(* CODESYS project contpiezasfun.project
   CustomField01_name: CustomField01
   CustomField08_name: CustomField08
   CustomField06_name: CustomField06
   Title: ATV_IMC_Template
   CustomField09_name: CustomField09
   CustomField07_name: CustomField07
   CustomField05_name: CustomField05
   Author: sergi gomez
   CustomField02_name: CustomField02
   Description: This template can be used for a correct interface with the local drive. the MANDATORY_AT_EACH_CYCLE program must be called like it is done in this application.
   CustomField04_name: CustomField04
   CustomField10_name: CustomField10
   Version: 0.0.0.0
   Company: Schneider Electric
   CustomField03_name: CustomField03

Project tree, tasks and I/O mapping:
  MyController : TM241CE24R, Schneider Electric, order no. TM241CE24R, version 4.0.2.9
    application Application
      task MAST (cyclic, interval 20 ms, priority 15, watchdog 100 ms x 1) calls progpiezas
      function HiddenPOU [ST]
      global variables GVL
      program progpiezas [LD]
      visualisation scada
    DI : Digital Inputs, Schneider Electric, version 4.0.2.9
        input  iwDI_IW0 : WORD  // IW0
        input  Application.progpiezas.sensorcil : BOOL  // IW0.I0
        input  Application.progpiezas.almacenaje : BOOL  // IW0.I1
        input  ibDI_IB1 : BYTE  // IB1
    DQ : Digital Outputs, Schneider Electric, version 4.0.2.9
        output qwDQ_QW0 : WORD  // QW0
        output qbDQ_QB1 : BYTE  // QB1
    Counters : Counters, Schneider Electric, version 4.0.2.9
    Pulse_Generators : Pulse Generators, Schneider Electric, version 4.0.2.9
    Cartridge_1 : Cartridge, Schneider Electric, version 4.0.2.9
    IO_Bus : IO bus - TM3, Schneider Electric, version 4.0.2.9
      Module_1 : TM3DQ8R/G, Schneider Electric, order no. TM3DQ8R/G, version 1.0.1.3
          output Application.progpiezas.contpiezas.cilrec : BOOL  // QB0.Q0
          output Application.progpiezas.contpiezas.cilext : BOOL  // QB0.Q1
          output Application.cinta : BOOL  // QB0.Q6
          unmapped channels: QB0
    COM_Bus : COM bus, Schneider Electric, version 4.0.2.9
    Ethernet_1 : Ethernet Network, Schneider Electric, version 4.0.2.9
    Serial_Line_1 : Serial line, Schneider Electric, version 4.0.2.9
      SoMachine_Network_Manager : SoMachine-Network Manager, Schneider Electric, version 4.0.0.2
    Serial_Line_2 : Serial line, Schneider Electric, version 4.0.2.9
      Modbus_Manager : Modbus Manager, Schneider Electric, version 4.0.0.2
  function block funcionpiezas [LD]
  text list GlobalTextList
*)

// MyController/Application/GVL
VAR_GLOBAL
	cinta: BOOL;
	marcha: BOOL;
END_VAR

// MyController/Application/progpiezas
PROGRAM progpiezas
VAR
	etapa0: BOOL;
	etapa1: BOOL;
	enviar: BOOL;
	etapa2: BOOL;
	contpiezas: funcionpiezas;
	almacenaje: BOOL;
	sensorcil: BOOL;
	piezauser: INT;
END_VAR
VAR_INPUT
	
END_VAR
VAR // added by the converter: edge detectors and wires of the graphical bodies
    _w1, _w2, _w3 : BOOL;
END_VAR

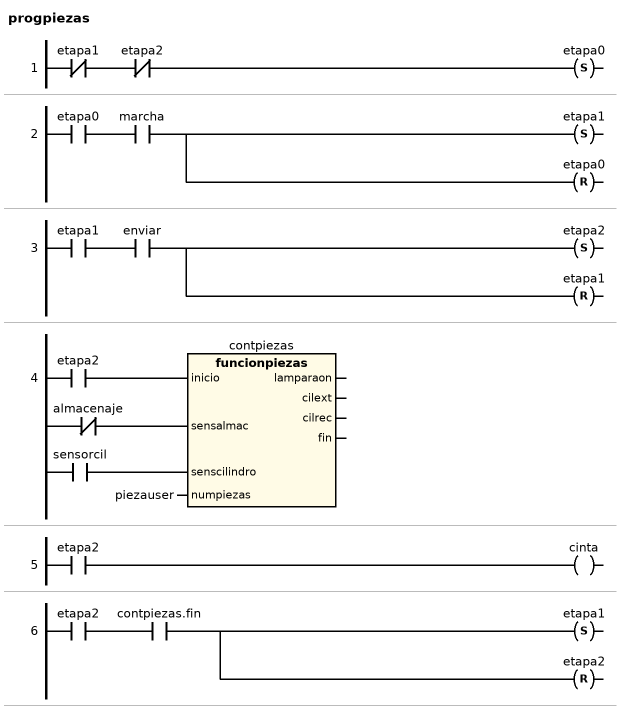
// NETWORK 1
etapa0 S= NOT etapa1 AND NOT etapa2;

// NETWORK 2
_w1 := etapa0 AND marcha;
etapa1 S= _w1;
etapa0 R= _w1;

// NETWORK 3
_w2 := etapa1 AND enviar;
etapa2 S= _w2;
etapa1 R= _w2;

// NETWORK 4
contpiezas(inicio := etapa2, sensalmac := NOT almacenaje, senscilindro := sensorcil, numpiezas := piezauser); // funcionpiezas

// NETWORK 5
cinta := etapa2;

// NETWORK 6
_w3 := etapa2 AND contpiezas.fin;
etapa1 S= _w3;
etapa2 R= _w3;

END_PROGRAM

// funcionpiezas
FUNCTION_BLOCK funcionpiezas
VAR_INPUT
	inicio: BOOL;
	
	sensalmac: BOOL;
	senscilindro: BOOL;
	numpiezas: INT;
END_VAR
VAR_OUTPUT
	lamparaon: BOOL;
	cilext: BOOL;
	cilrec: BOOL;
	fin: BOOL;
END_VAR
VAR
	etapa0: BOOL;
	
	etapa1: BOOL;
	espera: BOOL;
	etapa2: BOOL;
	tempo: TON;
	etapa3: BOOL;
	contpiezas: BOOL;
	etapa4: BOOL;
	
	
	tempcil: TON;
	contador: CTU;
END_VAR
VAR // added by the converter: edge detectors and wires of the graphical bodies
    _w1, _w2, _w3, _w4, _w5 : BOOL;
END_VAR

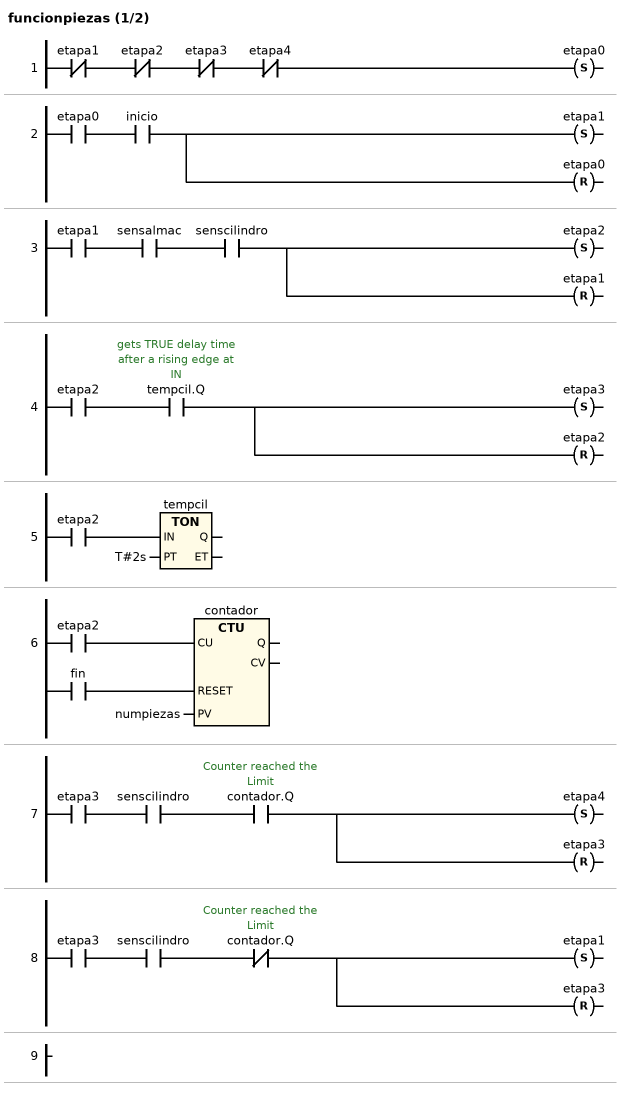
// NETWORK 1
etapa0 S= NOT etapa1 AND NOT etapa2 AND NOT etapa3 AND NOT etapa4;

// NETWORK 2
_w1 := etapa0 AND inicio;
etapa1 S= _w1;
etapa0 R= _w1;

// NETWORK 3
_w2 := etapa1 AND sensalmac AND senscilindro;
etapa2 S= _w2;
etapa1 R= _w2;

// NETWORK 4
//   tempcil.Q: gets TRUE delay time after a rising edge at IN
_w3 := etapa2 AND tempcil.Q;
etapa3 S= _w3;
etapa2 R= _w3;

// NETWORK 5
tempcil(IN := etapa2, PT := T#2s); // TON

// NETWORK 6
contador(CU := etapa2, RESET := fin, PV := numpiezas); // CTU

// NETWORK 7
//   contador.Q: Counter reached the Limit
_w4 := etapa3 AND senscilindro AND contador.Q;
etapa4 S= _w4;
etapa3 R= _w4;

// NETWORK 8
//   contador.Q: Counter reached the Limit
_w5 := etapa3 AND senscilindro AND NOT contador.Q;
etapa1 S= _w5;
etapa3 R= _w5;

// NETWORK 9

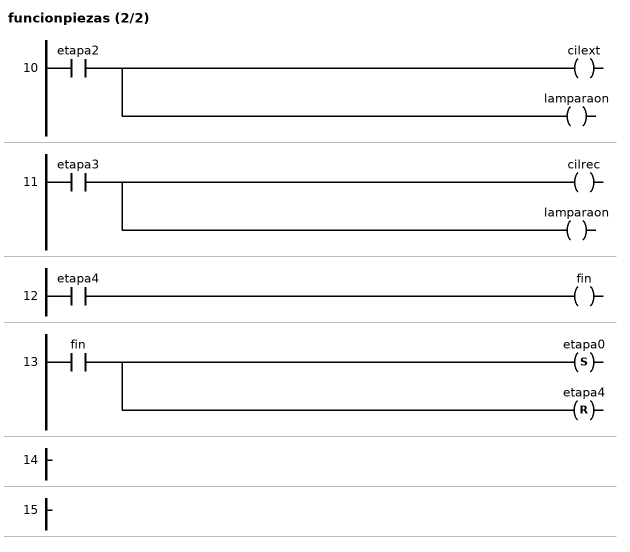
// NETWORK 10
cilext := etapa2;
lamparaon := etapa2;

// NETWORK 11
cilrec := etapa3;
lamparaon := etapa3;

// NETWORK 12
fin := etapa4;

// NETWORK 13
etapa0 S= fin;
etapa4 R= fin;

// NETWORK 14

// NETWORK 15

END_FUNCTION_BLOCK

// MyController/Application/HiddenPOU
FUNCTION HiddenPOU : BOOL

VAR_INPUT
	pHiddenFunc: POINTER TO WORD;
END_VAR
VAR
	pRead: POINTER TO BYTE;
	pWrite: POINTER TO BYTE;
END_VAR

pRead := pHiddenFunc + 400;
pWrite := pHiddenFunc + 4400;
HiddenPOU := TRUE;

END_FUNCTION

// MyController/Application/scada
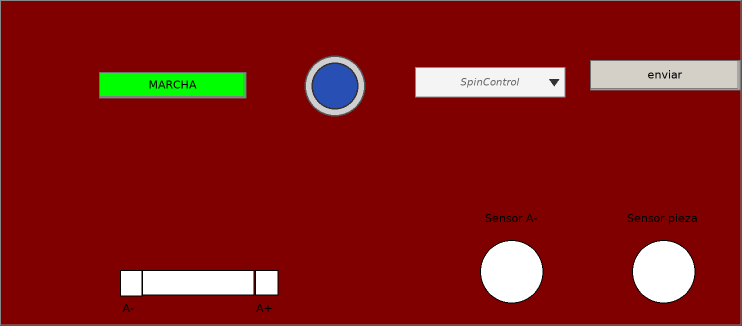
VISUALIZATION scada  // 742x326
    Button (99,72 147x26), "MARCHA"
        tap marcha
    Lamp1 (300,51 70x70), variable: progpiezas.contpiezas.lamparaon, style: Lamp-Lamp1-Blue
    SpinControl (415,67 150x30), variable: progpiezas.piezauser
    Button (590,60 150x30), "enviar"
        tap progpiezas.enviar
    Rectangle (255,270 23x25), colour toggle: progpiezas.contpiezas.cilext
    Rectangle (142,270 112x25)
    Label (106,293 45x31), "A-"
    Label (242,293 45x31), "A+"
    Ellipse (480,240 63x63), colour toggle: progpiezas.sensorcil
    Ellipse (632,240 63x63), colour toggle: progpiezas.almacenaje
        tap progpiezas.contpiezas.sensalmac p3779583253=TRUE
    Label (467,203 89x31), "Sensor A-"
    Label (618,203 89x31), "Sensor pieza"
    Rectangle (120,270 22x26), colour toggle: progpiezas.contpiezas.cilrec
END_VISUALIZATION
